// TIA Portal V20 export
TYPE "LER_typeUnitTrackingData"
// stored: Access Published
   STRUCT
      hotPressLeft { ExternalWritable := 'False'} : "LER_typeServoPressTrackingData";
      hotPressRight { ExternalWritable := 'False'} : "LER_typeServoPressTrackingData";
      hipotThicknesPress { S7_SetPoint := 'True'} : "LER_typeServoPressTrackingData";
      hipot { ExternalWritable := 'False'} : "LER_typeHipotTrackingData";
      thickness { ExternalWritable := 'False'} : "LER_typeThicknessTrackingData";
      vision { ExternalWritable := 'False'} : "LER_typeVisionTrackingData";
      laserMarker { ExternalWritable := 'False'} : "LER_typeMarkAndReadTrackingData";
      qrFixReader { ExternalWritable := 'False'} : "LER_typeMarkAndReadTrackingData";
      weightChecker { ExternalWritable := 'False'} : "LER_typeWeightCheckTrackingData";
      markAndReadCompare { ExternalWritable := 'False'} : Bool;   // 0: NG, 1: OK
   END_STRUCT;
END_TYPE
